PROGRAM MAIN
VAR
	bAddEvent : BOOL;
	rtrigAddEvent : R_TRIG;
	
	eEventType : E_EventType := E_EventType.Alarm;
	eEventSeverity : TcEventSeverity := TcEventSeverity.Error;
	nEventIdentity : UDINT := 42;;
	sEventText : STRING(255) := 'This is a scary event.';
	
	fbEventLogger : FB_EventLogger;
END_VAR


rtrigAddEvent(CLK := bAddEvent);

IF rtrigAddEvent.Q THEN
	fbEventLogger.AddEvent(
		eEventType:= eEventType,
		eEventSeverity:= eEventSeverity,
		nEventIdentity:= nEventIdentity,
		sEventText:= sEventText);
END_IF

END_PROGRAM

(* stored: Version 1.1.0.1, ProductVersion 3.1.4024.15
   POU MAIN: Id {76ea4639-ff90-43ac-8456-dc4de8ad42a3}, SpecialFunc None *)
